TEXTLIST LineClose
  0 = 'LineCose_None'
  1 = 'LineClose_Line2'
  2 = 'LineClose_Line3'
   = ''
END_TEXTLIST

(* stored: Version 1.1.0.1, ProductVersion 3.1.4024.3
   TextList LineClose: Id {4638bc6c-f4e8-4ca1-b642-295b7dd6f40a} *)
